{attribute 'GeneratedUsingTerminal: EL3443-0000-0016'}
{attribute addProperty BoxType "EL3443-0000-0016"}
{attribute addProperty Id "VoltageAT %I*REAL4CurrentAT %I*REAL4"}
{attribute addProperty CRC "1717073118"}
{attribute addProperty Size "8"}
TYPE L2_Basic_665874DE EXTENDS InputBase_8311D824 :
STRUCT
	{attribute addProperty Name "Voltage"}
	Voltage AT %I* : REAL;
	{attribute addProperty Name "Current"}
	Current AT %I* : REAL;
END_STRUCT
END_TYPE

(* stored: Version 1.2.0.0, ProductVersion 3.1.4024.11
   DUT L2_Basic_665874DE: Id {e5fa05ba-5887-487f-97a5-ba243bb4cda3} *)
